// TwinCAT 3 PLC project PLC1
// ProgramVersion: 3.1.4024.0
// libraries:
//   Tc2_Standard, * (Beckhoff Automation GmbH)
//   Tc2_System, * (Beckhoff Automation GmbH)
//   Tc2_Utilities, * (Beckhoff Automation GmbH)
//   Tc3_Module, * (Beckhoff Automation GmbH)
// project tree:
//   / PlcTask.TcTTO
//   POUs/FBs/ FB_Clock.TcPOU (not stored)
//   POUs/ MAIN.TcPOU, P_LubLogic.TcPOU
// real-time tasks:
//   TASK PlcTask: cycle T#10ms, priority 20, ADS port 350

CONFIGURATION PLC1
    RESOURCE PLC ON TwinCAT3
        TASK PlcTask(INTERVAL := T#10ms, PRIORITY := 20);
        PROGRAM MAIN WITH PlcTask : MAIN;
    END_RESOURCE
END_CONFIGURATION

// ---- POUs/MAIN.TcPOU
PROGRAM MAIN
VAR
	fbWritePersistentData	: FB_WritePersistentData; (* Chamada do bloco para salvar variáveis persistentes*)
	fbClock					: FB_CLOCK; (* Bloco CLOCK *)
END_VAR

ACT_Persistent(); (* Action com os blocos persistentes *)

P_LubLogic(); (* Lógica de Lubrificação *)

ACTION ACT_Persistent:
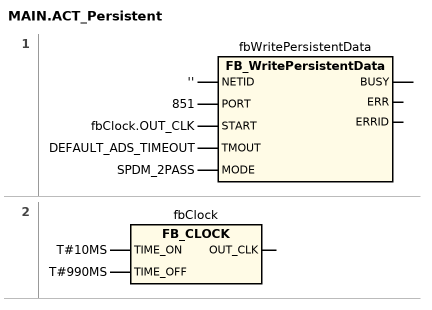
// NETWORK 1
fbWritePersistentData(
    NETID := '',
    PORT := 851,
    START := fbClock.OUT_CLK,
    TMOUT := DEFAULT_ADS_TIMEOUT,
    MODE := SPDM_2PASS); // FB_WritePersistentData

// NETWORK 2
fbClock(TIME_ON := T#10MS, TIME_OFF := T#990MS); // FB_CLOCK
END_ACTION

END_PROGRAM

// ---- POUs/P_LubLogic.TcPOU
PROGRAM P_LubLogic
VAR
	TON_MaqLigada 			: TON;
	bMaquinaLigada			: BOOL;
	tEsperaLubrificacao		: TIME := T#30S;
	tLubrificacao			: TIME := T#5S;
	TON_Lubrificando		: TON;
	bFirstScan				: BOOL := TRUE;
	doLubrificacao			: BOOL;
	tiSoma					: TIME;	
	tiSomaOdometro			: TIME;	
END_VAR

VAR PERSISTENT	
	tiOdometro				: TIME;
	tiOdometro_Old			: TIME;
END_VAR
VAR // added by the converter: edge detectors and wires of the graphical bodies
    _w1 : BOOL;
END_VAR

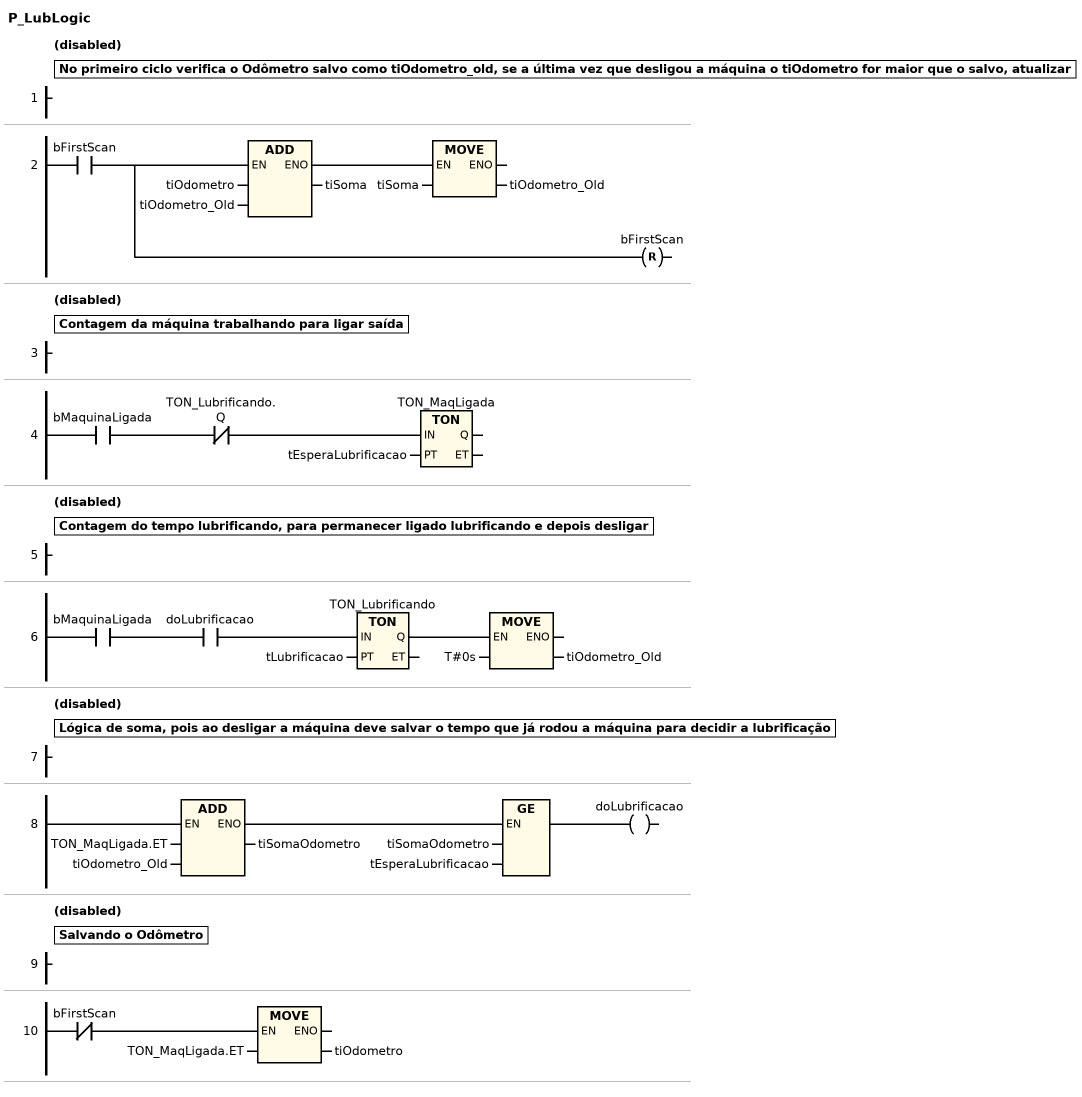
// NETWORK 1 (disabled)
// label: No primeiro ciclo verifica o Odômetro salvo como tiOdometro_old, se a última vez que desligou a máquina o tiOdometro for maior que o salvo, atualizar

// NETWORK 2
_w1 := bFirstScan;
IF _w1 THEN tiSoma := tiOdometro + tiOdometro_Old; END_IF
IF _w1 THEN tiOdometro_Old := tiSoma; END_IF
bFirstScan R= _w1;

// NETWORK 3 (disabled)
// label: Contagem da máquina trabalhando para ligar saída

// NETWORK 4
TON_MaqLigada(IN := bMaquinaLigada AND NOT TON_Lubrificando.Q, PT := tEsperaLubrificacao); // TON

// NETWORK 5 (disabled)
// label: Contagem do tempo lubrificando, para permanecer ligado lubrificando e depois desligar

// NETWORK 6
TON_Lubrificando(IN := bMaquinaLigada AND doLubrificacao, PT := tLubrificacao); // TON
IF TON_Lubrificando.Q THEN tiOdometro_Old := T#0s; END_IF

// NETWORK 7 (disabled)
// label: Lógica de soma, pois ao desligar a máquina deve salvar o tempo que já rodou a máquina para decidir a lubrificação

// NETWORK 8
tiSomaOdometro := TON_MaqLigada.ET + tiOdometro_Old;
doLubrificacao := tiSomaOdometro >= tEsperaLubrificacao;

// NETWORK 9 (disabled)
// label: Salvando o Odômetro

// NETWORK 10
IF NOT bFirstScan THEN tiOdometro := TON_MaqLigada.ET; END_IF

END_PROGRAM
